// TIA Portal V18 export
FUNCTION "Function Selection HMI _Site_PB" : Void   // FC30, LAD
{ S7_Optimized_Access := 'TRUE' }
VERSION : 0.1
// stored: AutoNumber true, IsIECCheckEnabled false, SetENOAutomatically false, UDAEnableTagReadback false
   VAR_TEMP
      temp_unitsel : Int;
   END_VAR
   VAR_TEMP   // added for the SCL form of the ladder/FBD networks
      _w1 : Bool;
      _w2 : Bool;
   END_VAR
BEGIN

REGION Network 1: No functions selected
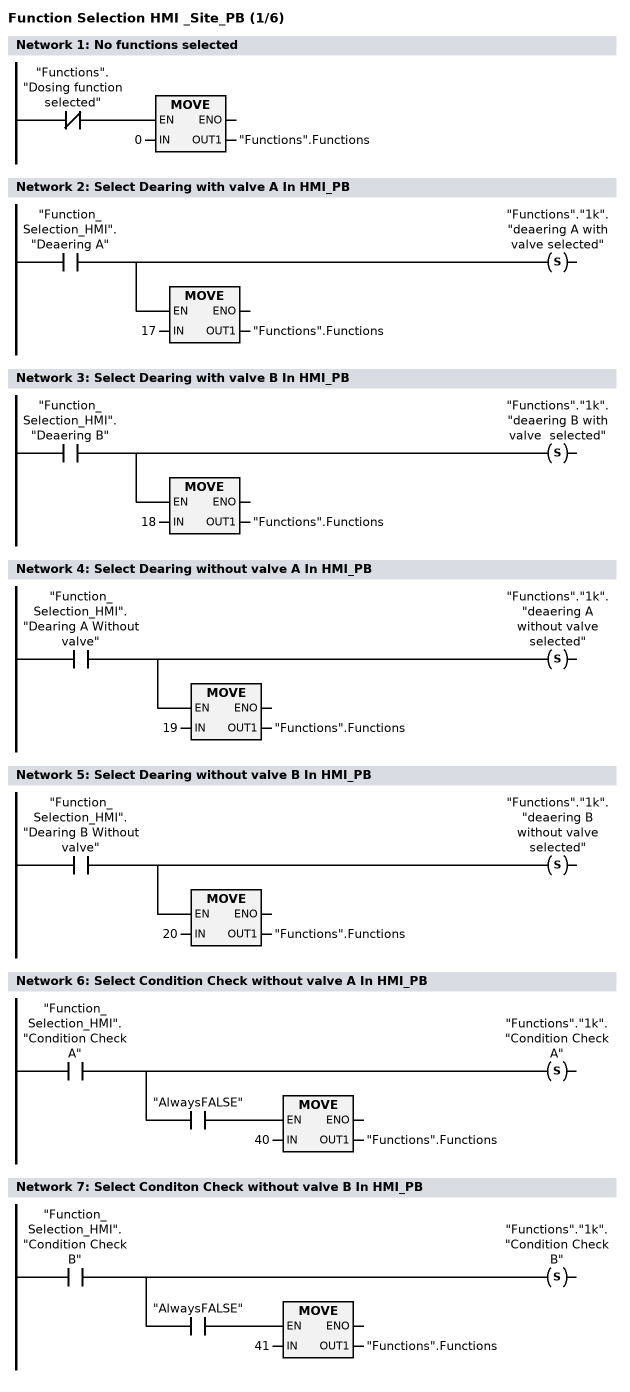
   RUNG wire#powerrail
      I_Contact( "Functions"."Dosing function selected" )
      Move(in := 0, out1 => "Functions".Functions)
   END_RUNG
   // the same network as SCL:
   IF NOT "Functions"."Dosing function selected" THEN "Functions".Functions := 0; END_IF;
END_REGION

REGION Network 2: Select Dearing with valve A In HMI_PB
   RUNG wire#powerrail
      Contact( "Function_Selection_HMI"."Deaering A" )
      wire#w1
      S_Coil( "Functions"."1k"."deaering A with valve selected" )
   END_RUNG
   RUNG wire#w1
      Move(in := 17, out1 => "Functions".Functions)
   END_RUNG
   // the same network as SCL:
   IF "Function_Selection_HMI"."Deaering A" THEN
       "Functions"."1k"."deaering A with valve selected" := TRUE;
       "Functions".Functions := 17;
   END_IF;
END_REGION

REGION Network 3: Select Dearing with valve B In HMI_PB
   RUNG wire#powerrail
      Contact( "Function_Selection_HMI"."Deaering B" )
      wire#w1
      S_Coil( "Functions"."1k"."deaering B with valve  selected" )
   END_RUNG
   RUNG wire#w1
      Move(in := 18, out1 => "Functions".Functions)
   END_RUNG
   // the same network as SCL:
   IF "Function_Selection_HMI"."Deaering B" THEN
       "Functions"."1k"."deaering B with valve  selected" := TRUE;
       "Functions".Functions := 18;
   END_IF;
END_REGION

REGION Network 4: Select Dearing without valve A In HMI_PB
   RUNG wire#powerrail
      Contact( "Function_Selection_HMI"."Dearing A Without valve" )
      wire#w1
      S_Coil( "Functions"."1k"."deaering A without valve selected" )
   END_RUNG
   RUNG wire#w1
      Move(in := 19, out1 => "Functions".Functions)
   END_RUNG
   // the same network as SCL:
   IF "Function_Selection_HMI"."Dearing A Without valve" THEN
       "Functions"."1k"."deaering A without valve selected" := TRUE;
       "Functions".Functions := 19;
   END_IF;
END_REGION

REGION Network 5: Select Dearing without valve B In HMI_PB
   RUNG wire#powerrail
      Contact( "Function_Selection_HMI"."Dearing B Without valve" )
      wire#w1
      S_Coil( "Functions"."1k"."deaering B without valve  selected" )
   END_RUNG
   RUNG wire#w1
      Move(in := 20, out1 => "Functions".Functions)
   END_RUNG
   // the same network as SCL:
   IF "Function_Selection_HMI"."Dearing B Without valve" THEN
       "Functions"."1k"."deaering B without valve  selected" := TRUE;
       "Functions".Functions := 20;
   END_IF;
END_REGION

REGION Network 6: Select Condition Check without valve A In HMI_PB
   RUNG wire#powerrail
      Contact( "Function_Selection_HMI"."Condition Check A" )
      wire#w1
      S_Coil( "Functions"."1k"."Condition Check A" )
   END_RUNG
   RUNG wire#w1
      Contact( "AlwaysFALSE" )
      Move(in := 40, out1 => "Functions".Functions)
   END_RUNG
   // the same network as SCL:
   IF "Function_Selection_HMI"."Condition Check A" THEN "Functions"."1k"."Condition Check A" := TRUE; END_IF;
   IF "Function_Selection_HMI"."Condition Check A" AND "AlwaysFALSE" THEN
       "Functions".Functions := 40;
   END_IF;
END_REGION

REGION Network 7: Select Conditon Check without valve B In HMI_PB
   RUNG wire#powerrail
      Contact( "Function_Selection_HMI"."Condition Check B" )
      wire#w1
      S_Coil( "Functions"."1k"."Condition Check B" )
   END_RUNG
   RUNG wire#w1
      Contact( "AlwaysFALSE" )
      Move(in := 41, out1 => "Functions".Functions)
   END_RUNG
   // the same network as SCL:
   IF "Function_Selection_HMI"."Condition Check B" THEN "Functions"."1k"."Condition Check B" := TRUE; END_IF;
   IF "Function_Selection_HMI"."Condition Check B" AND "AlwaysFALSE" THEN
       "Functions".Functions := 41;
   END_IF;
END_REGION

REGION Network 8: Select Recirculation A
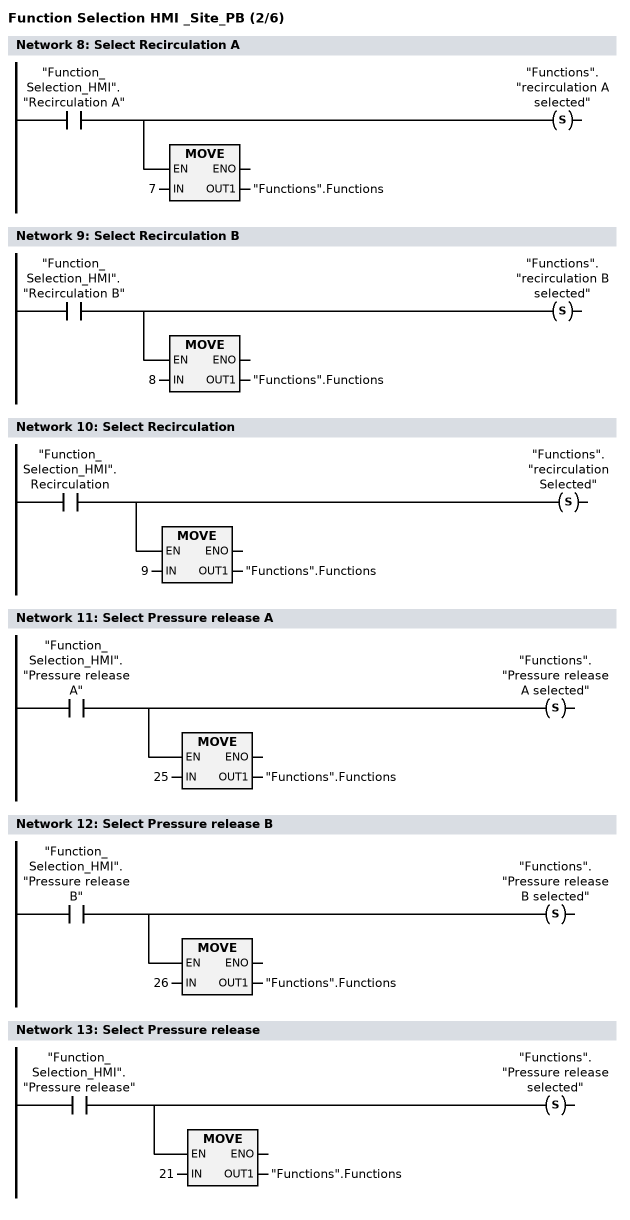
   RUNG wire#powerrail
      Contact( "Function_Selection_HMI"."Recirculation A" )
      wire#w1
      S_Coil( "Functions"."recirculation A selected" )
   END_RUNG
   RUNG wire#w1
      Move(in := 7, out1 => "Functions".Functions)
   END_RUNG
   // the same network as SCL:
   IF "Function_Selection_HMI"."Recirculation A" THEN
       "Functions"."recirculation A selected" := TRUE;
       "Functions".Functions := 7;
   END_IF;
END_REGION

REGION Network 9: Select Recirculation B
   RUNG wire#powerrail
      Contact( "Function_Selection_HMI"."Recirculation B" )
      wire#w1
      S_Coil( "Functions"."recirculation B selected" )
   END_RUNG
   RUNG wire#w1
      Move(in := 8, out1 => "Functions".Functions)
   END_RUNG
   // the same network as SCL:
   IF "Function_Selection_HMI"."Recirculation B" THEN
       "Functions"."recirculation B selected" := TRUE;
       "Functions".Functions := 8;
   END_IF;
END_REGION

REGION Network 10: Select Recirculation
   RUNG wire#powerrail
      Contact( "Function_Selection_HMI".Recirculation )
      wire#w1
      S_Coil( "Functions"."recirculation Selected" )
   END_RUNG
   RUNG wire#w1
      Move(in := 9, out1 => "Functions".Functions)
   END_RUNG
   // the same network as SCL:
   IF "Function_Selection_HMI".Recirculation THEN
       "Functions"."recirculation Selected" := TRUE;
       "Functions".Functions := 9;
   END_IF;
END_REGION

REGION Network 11: Select Pressure release A
   RUNG wire#powerrail
      Contact( "Function_Selection_HMI"."Pressure release A" )
      wire#w1
      S_Coil( "Functions"."Pressure release A selected" )
   END_RUNG
   RUNG wire#w1
      Move(in := 25, out1 => "Functions".Functions)
   END_RUNG
   // the same network as SCL:
   IF "Function_Selection_HMI"."Pressure release A" THEN
       "Functions"."Pressure release A selected" := TRUE;
       "Functions".Functions := 25;
   END_IF;
END_REGION

REGION Network 12: Select Pressure release B
   RUNG wire#powerrail
      Contact( "Function_Selection_HMI"."Pressure release B" )
      wire#w1
      S_Coil( "Functions"."Pressure release B selected" )
   END_RUNG
   RUNG wire#w1
      Move(in := 26, out1 => "Functions".Functions)
   END_RUNG
   // the same network as SCL:
   IF "Function_Selection_HMI"."Pressure release B" THEN
       "Functions"."Pressure release B selected" := TRUE;
       "Functions".Functions := 26;
   END_IF;
END_REGION

REGION Network 13: Select Pressure release
   RUNG wire#powerrail
      Contact( "Function_Selection_HMI"."Pressure release" )
      wire#w1
      S_Coil( "Functions"."Pressure release selected" )
   END_RUNG
   RUNG wire#w1
      Move(in := 21, out1 => "Functions".Functions)
   END_RUNG
   // the same network as SCL:
   IF "Function_Selection_HMI"."Pressure release" THEN
       "Functions"."Pressure release selected" := TRUE;
       "Functions".Functions := 21;
   END_IF;
END_REGION

REGION Network 14: Select shot metering
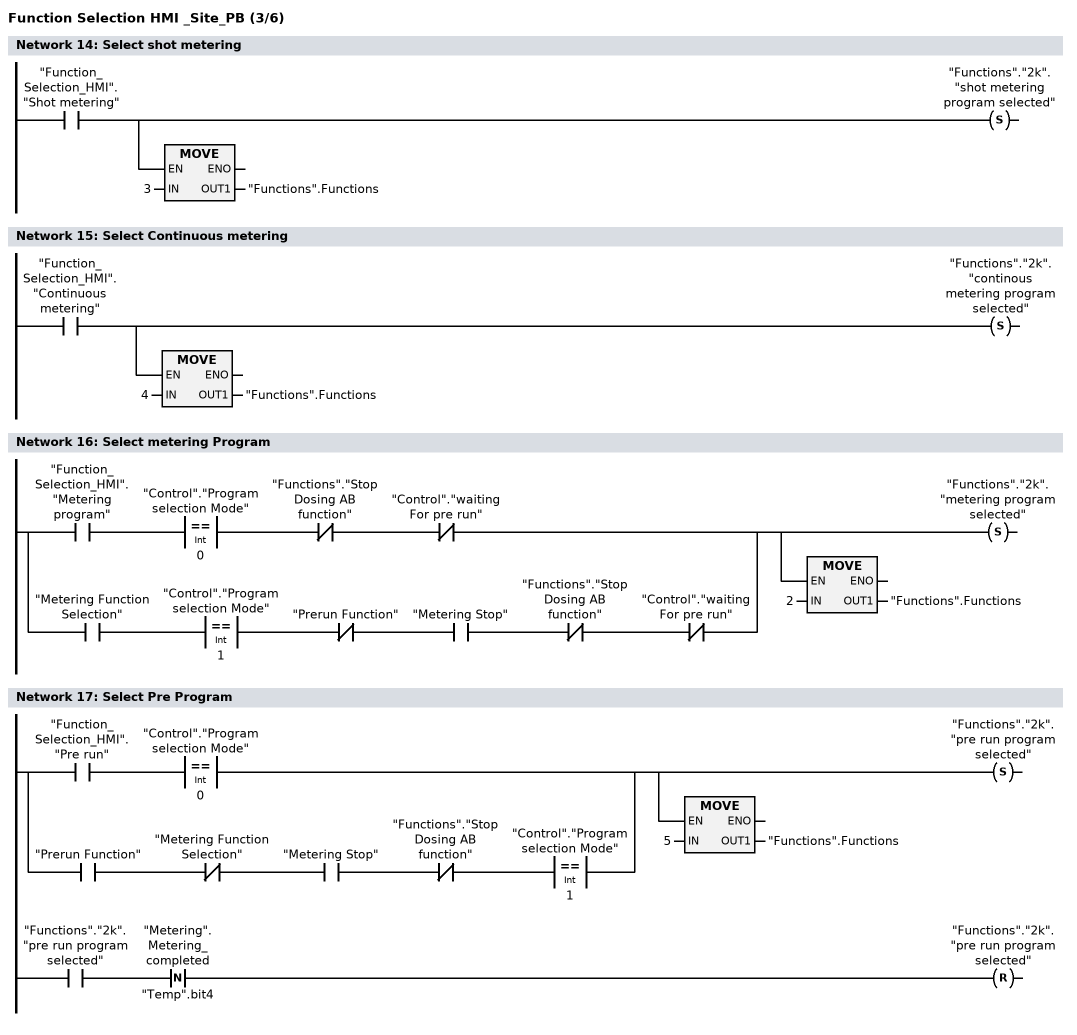
   RUNG wire#powerrail
      Contact( "Function_Selection_HMI"."Shot metering" )
      wire#w1
      S_Coil( "Functions"."2k"."shot metering program selected" )
   END_RUNG
   RUNG wire#w1
      Move(in := 3, out1 => "Functions".Functions)
   END_RUNG
   // the same network as SCL:
   IF "Function_Selection_HMI"."Shot metering" THEN
       "Functions"."2k"."shot metering program selected" := TRUE;
       "Functions".Functions := 3;
   END_IF;
END_REGION

REGION Network 15: Select Continuous metering
   RUNG wire#powerrail
      Contact( "Function_Selection_HMI"."Continuous metering" )
      wire#w1
      S_Coil( "Functions"."2k"."continous metering program selected" )
   END_RUNG
   RUNG wire#w1
      Move(in := 4, out1 => "Functions".Functions)
   END_RUNG
   // the same network as SCL:
   IF "Function_Selection_HMI"."Continuous metering" THEN
       "Functions"."2k"."continous metering program selected" := TRUE;
       "Functions".Functions := 4;
   END_IF;
END_REGION

REGION Network 16: Select metering Program
   RUNG wire#powerrail
      Contact( "Function_Selection_HMI"."Metering program" )
      { S7_Templates := "SrcType := Int" } EQ_Contact(in1 := "Control"."Program selection Mode", in2 := 0)
      I_Contact( "Functions"."Stop Dosing AB function" )
      I_Contact( "Control"."waiting For pre run" )
      wire#w1
      S_Coil( "Functions"."2k"."metering program selected" )
   END_RUNG
   RUNG wire#powerrail
      Contact( "Metering Function Selection" )
      { S7_Templates := "SrcType := Int" } EQ_Contact(in1 := "Control"."Program selection Mode", in2 := 1)
      I_Contact( "Prerun Function" )
      Contact( "Metering Stop" )
      I_Contact( "Functions"."Stop Dosing AB function" )
      I_Contact( "Control"."waiting For pre run" )
   END_RUNG wire#w1
   RUNG wire#w1
      Move(in := 2, out1 => "Functions".Functions)
   END_RUNG
   // the same network as SCL:
   IF ("Function_Selection_HMI"."Metering program" AND ("Control"."Program selection Mode" = 0) AND NOT "Functions"."Stop Dosing AB function" AND NOT "Control"."waiting For pre run") OR ("Metering Function Selection" AND ("Control"."Program selection Mode" = 1) AND NOT "Prerun Function" AND "Metering Stop" AND NOT "Functions"."Stop Dosing AB function" AND NOT "Control"."waiting For pre run") THEN
       "Functions"."2k"."metering program selected" := TRUE;
       "Functions".Functions := 2;
   END_IF;
END_REGION

REGION Network 17: Select Pre Program
   RUNG wire#powerrail
      Contact( "Function_Selection_HMI"."Pre run" )
      { S7_Templates := "SrcType := Int" } EQ_Contact(in1 := "Control"."Program selection Mode", in2 := 0)
      wire#w1
      S_Coil( "Functions"."2k"."pre run program selected" )
   END_RUNG
   RUNG wire#powerrail
      Contact( "Prerun Function" )
      I_Contact( "Metering Function Selection" )
      Contact( "Metering Stop" )
      I_Contact( "Functions"."Stop Dosing AB function" )
      { S7_Templates := "SrcType := Int" } EQ_Contact(in1 := "Control"."Program selection Mode", in2 := 1)
   END_RUNG wire#w1
   RUNG wire#w1
      Move(in := 5, out1 => "Functions".Functions)
   END_RUNG
   RUNG wire#powerrail
      Contact( "Functions"."2k"."pre run program selected" )
      N_Contact(operand := "Metering".Metering_completed, bit := "Temp".bit4)
      R_Coil( "Functions"."2k"."pre run program selected" )
   END_RUNG
   // the same network as SCL:
   IF ("Function_Selection_HMI"."Pre run" AND ("Control"."Program selection Mode" = 0)) OR ("Prerun Function" AND NOT "Metering Function Selection" AND "Metering Stop" AND NOT "Functions"."Stop Dosing AB function" AND ("Control"."Program selection Mode" = 1)) THEN
       "Functions"."2k"."pre run program selected" := TRUE;
       "Functions".Functions := 5;
   END_IF;
   #_w1 := "Functions"."2k"."pre run program selected" AND NOT "Metering".Metering_completed AND "Temp".bit4;   // falling edge of "Metering".Metering_completed
   "Temp".bit4 := "Metering".Metering_completed;
   IF #_w1 THEN "Functions"."2k"."pre run program selected" := FALSE; END_IF;
END_REGION

REGION Network 18: Select Ratio Program
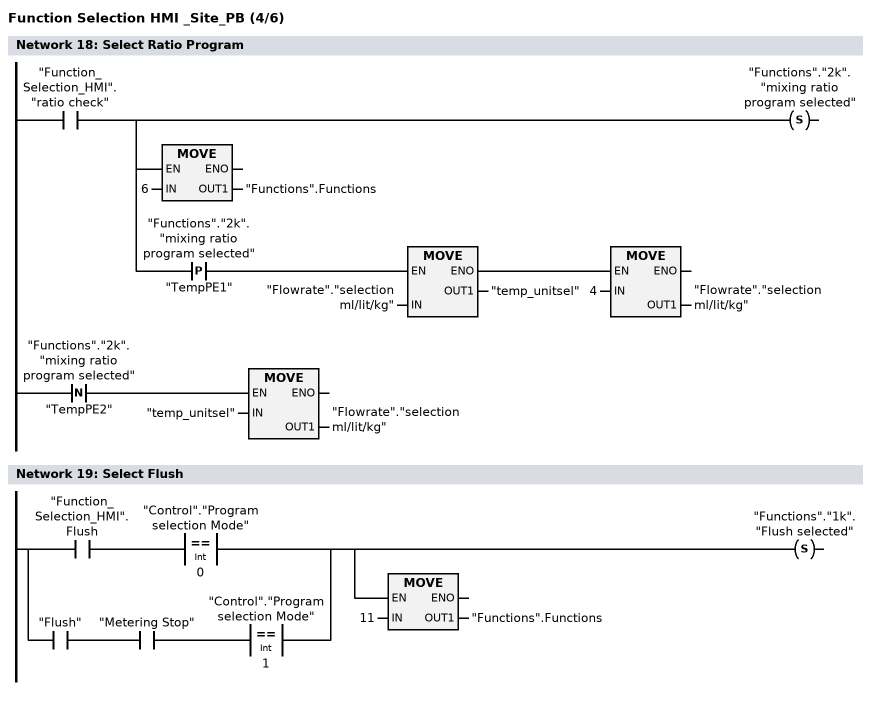
   RUNG wire#powerrail
      Contact( "Function_Selection_HMI"."ratio check" )
      wire#w1
      S_Coil( "Functions"."2k"."mixing ratio program selected" )
   END_RUNG
   RUNG wire#w1
      Move(in := 6, out1 => "Functions".Functions)
   END_RUNG
   RUNG wire#w1
      P_Contact(operand := "Functions"."2k"."mixing ratio program selected", bit := "TempPE1")
      Move(in := "Flowrate"."selection ml/lit/kg", out1 => "temp_unitsel")
      Move(in := 4, out1 => "Flowrate"."selection ml/lit/kg")
   END_RUNG
   RUNG wire#powerrail
      N_Contact(operand := "Functions"."2k"."mixing ratio program selected", bit := "TempPE2")
      Move(in := "temp_unitsel", out1 => "Flowrate"."selection ml/lit/kg")
   END_RUNG
   // the same network as SCL:
   IF "Function_Selection_HMI"."ratio check" THEN
       "Functions"."2k"."mixing ratio program selected" := TRUE;
       "Functions".Functions := 6;
   END_IF;
   #_w1 := "Function_Selection_HMI"."ratio check" AND "Functions"."2k"."mixing ratio program selected" AND NOT "TempPE1";   // rising edge of "Functions"."2k"."mixing ratio program selected"
   "TempPE1" := "Functions"."2k"."mixing ratio program selected";
   IF #_w1 THEN
       "temp_unitsel" := "Flowrate"."selection ml/lit/kg";
       "Flowrate"."selection ml/lit/kg" := 4;
   END_IF;
   #_w2 := NOT "Functions"."2k"."mixing ratio program selected" AND "TempPE2";   // falling edge of "Functions"."2k"."mixing ratio program selected"
   "TempPE2" := "Functions"."2k"."mixing ratio program selected";
   IF #_w2 THEN "Flowrate"."selection ml/lit/kg" := "temp_unitsel"; END_IF;
END_REGION

REGION Network 19: Select Flush
   RUNG wire#powerrail
      Contact( "Function_Selection_HMI".Flush )
      { S7_Templates := "SrcType := Int" } EQ_Contact(in1 := "Control"."Program selection Mode", in2 := 0)
      wire#w1
      S_Coil( "Functions"."1k"."Flush selected" )
   END_RUNG
   RUNG wire#powerrail
      Contact( "Flush" )
      Contact( "Metering Stop" )
      { S7_Templates := "SrcType := Int" } EQ_Contact(in1 := "Control"."Program selection Mode", in2 := 1)
   END_RUNG wire#w1
   RUNG wire#w1
      Move(in := 11, out1 => "Functions".Functions)
   END_RUNG
   // the same network as SCL:
   IF ("Function_Selection_HMI".Flush AND ("Control"."Program selection Mode" = 0)) OR ("Flush" AND "Metering Stop" AND ("Control"."Program selection Mode" = 1)) THEN
       "Functions"."1k"."Flush selected" := TRUE;
       "Functions".Functions := 11;
   END_IF;
END_REGION

REGION Network 20: Select Flush during potlife
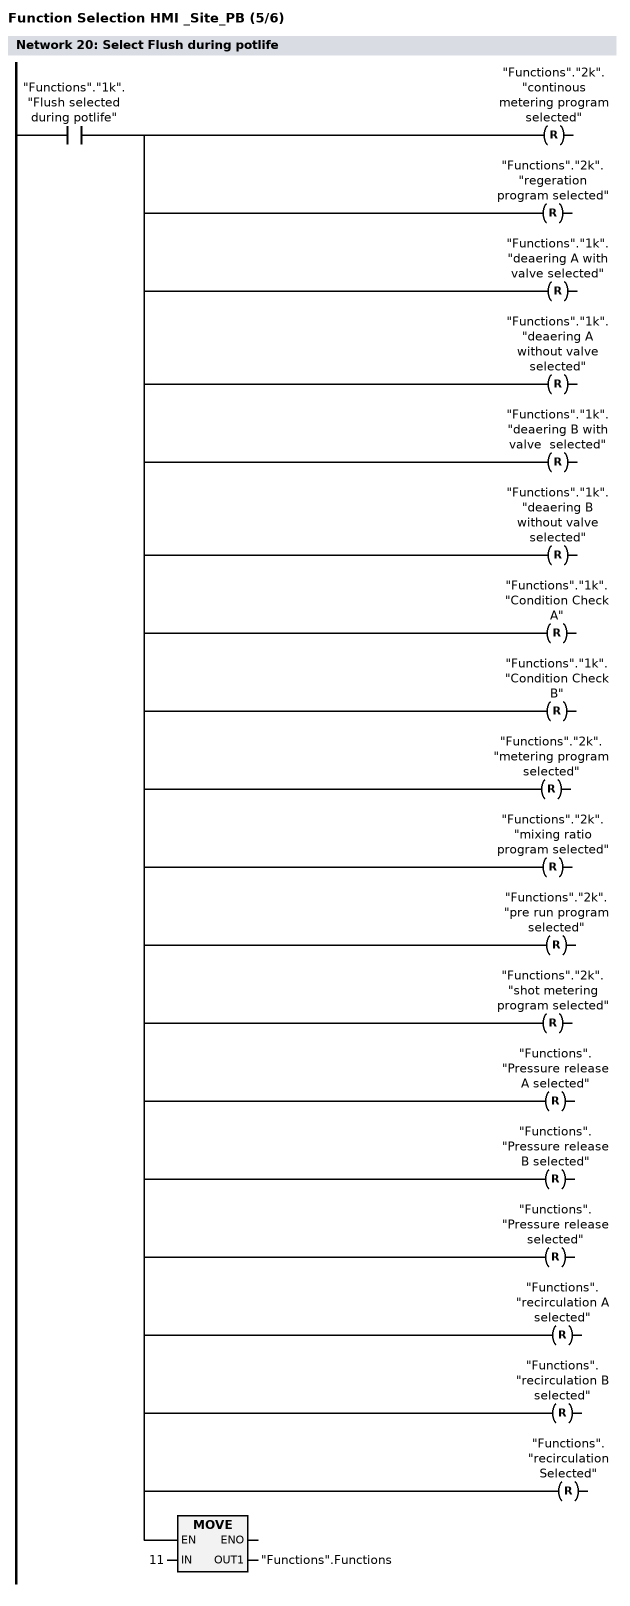
   RUNG wire#powerrail
      Contact( "Functions"."1k"."Flush selected during potlife" )
      wire#w1
      R_Coil( "Functions"."2k"."continous metering program selected" )
   END_RUNG
   RUNG wire#w1
      R_Coil( "Functions"."2k"."regeration program selected" )
   END_RUNG
   RUNG wire#w1
      R_Coil( "Functions"."1k"."deaering A with valve selected" )
   END_RUNG
   RUNG wire#w1
      R_Coil( "Functions"."1k"."deaering A without valve selected" )
   END_RUNG
   RUNG wire#w1
      R_Coil( "Functions"."1k"."deaering B with valve  selected" )
   END_RUNG
   RUNG wire#w1
      R_Coil( "Functions"."1k"."deaering B without valve  selected" )
   END_RUNG
   RUNG wire#w1
      R_Coil( "Functions"."1k"."Condition Check A" )
   END_RUNG
   RUNG wire#w1
      R_Coil( "Functions"."1k"."Condition Check B" )
   END_RUNG
   RUNG wire#w1
      R_Coil( "Functions"."2k"."metering program selected" )
   END_RUNG
   RUNG wire#w1
      R_Coil( "Functions"."2k"."mixing ratio program selected" )
   END_RUNG
   RUNG wire#w1
      R_Coil( "Functions"."2k"."pre run program selected" )
   END_RUNG
   RUNG wire#w1
      R_Coil( "Functions"."2k"."shot metering program selected" )
   END_RUNG
   RUNG wire#w1
      R_Coil( "Functions"."Pressure release A selected" )
   END_RUNG
   RUNG wire#w1
      R_Coil( "Functions"."Pressure release B selected" )
   END_RUNG
   RUNG wire#w1
      R_Coil( "Functions"."Pressure release selected" )
   END_RUNG
   RUNG wire#w1
      R_Coil( "Functions"."recirculation A selected" )
   END_RUNG
   RUNG wire#w1
      R_Coil( "Functions"."recirculation B selected" )
   END_RUNG
   RUNG wire#w1
      R_Coil( "Functions"."recirculation Selected" )
   END_RUNG
   RUNG wire#w1
      Move(in := 11, out1 => "Functions".Functions)
   END_RUNG
   // the same network as SCL:
   IF "Functions"."1k"."Flush selected during potlife" THEN
       "Functions"."2k"."continous metering program selected" := FALSE;
       "Functions"."2k"."regeration program selected" := FALSE;
       "Functions"."1k"."deaering A with valve selected" := FALSE;
       "Functions"."1k"."deaering A without valve selected" := FALSE;
       "Functions"."1k"."deaering B with valve  selected" := FALSE;
       "Functions"."1k"."deaering B without valve  selected" := FALSE;
       "Functions"."1k"."Condition Check A" := FALSE;
       "Functions"."1k"."Condition Check B" := FALSE;
       "Functions"."2k"."metering program selected" := FALSE;
       "Functions"."2k"."mixing ratio program selected" := FALSE;
       "Functions"."2k"."pre run program selected" := FALSE;
       "Functions"."2k"."shot metering program selected" := FALSE;
       "Functions"."Pressure release A selected" := FALSE;
       "Functions"."Pressure release B selected" := FALSE;
       "Functions"."Pressure release selected" := FALSE;
       "Functions"."recirculation A selected" := FALSE;
       "Functions"."recirculation B selected" := FALSE;
       "Functions"."recirculation Selected" := FALSE;
       "Functions".Functions := 11;
   END_IF;
END_REGION

REGION Network 21: regeneration selected
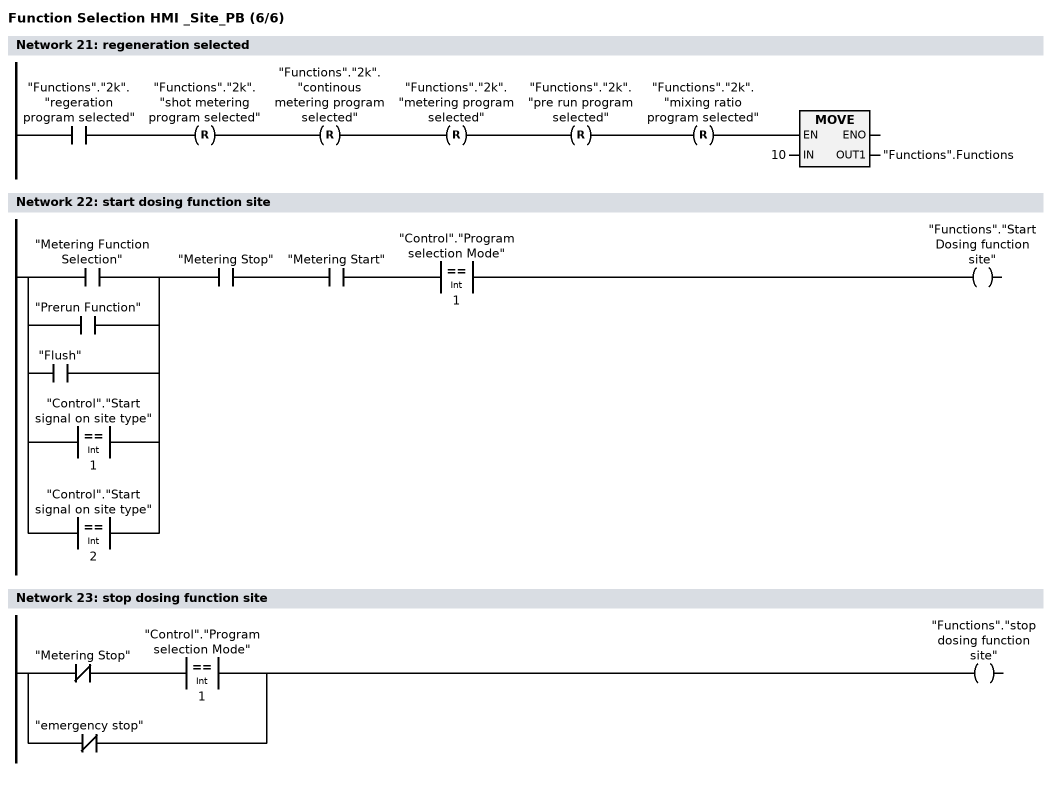
   RUNG wire#powerrail
      Contact( "Functions"."2k"."regeration program selected" )
      R_Coil( "Functions"."2k"."shot metering program selected" )
      R_Coil( "Functions"."2k"."continous metering program selected" )
      R_Coil( "Functions"."2k"."metering program selected" )
      R_Coil( "Functions"."2k"."pre run program selected" )
      R_Coil( "Functions"."2k"."mixing ratio program selected" )
      Move(in := 10, out1 => "Functions".Functions)
   END_RUNG
   // the same network as SCL:
   IF "Functions"."2k"."regeration program selected" THEN
       "Functions"."2k"."shot metering program selected" := FALSE;
       "Functions"."2k"."continous metering program selected" := FALSE;
       "Functions"."2k"."metering program selected" := FALSE;
       "Functions"."2k"."pre run program selected" := FALSE;
       "Functions"."2k"."mixing ratio program selected" := FALSE;
       "Functions".Functions := 10;
   END_IF;
END_REGION

REGION Network 22: start dosing function site
   RUNG wire#powerrail
      Contact( "Metering Function Selection" )
      wire#w1
      Contact( "Metering Stop" )
      Contact( "Metering Start" )
      { S7_Templates := "SrcType := Int" } EQ_Contact(in1 := "Control"."Program selection Mode", in2 := 1)
      Coil( "Functions"."Start Dosing function site" )
   END_RUNG
   RUNG wire#powerrail
      Contact( "Prerun Function" )
   END_RUNG wire#w1
   RUNG wire#powerrail
      Contact( "Flush" )
   END_RUNG wire#w1
   RUNG wire#powerrail
      { S7_Templates := "SrcType := Int" } EQ_Contact(in1 := "Control"."Start signal on site type", in2 := 1)
   END_RUNG wire#w1
   RUNG wire#powerrail
      { S7_Templates := "SrcType := Int" } EQ_Contact(in1 := "Control"."Start signal on site type", in2 := 2)
   END_RUNG wire#w1
   // the same network as SCL:
   "Functions"."Start Dosing function site" := ("Metering Function Selection" OR "Prerun Function" OR "Flush" OR ("Control"."Start signal on site type" = 1) OR ("Control"."Start signal on site type" = 2)) AND "Metering Stop" AND "Metering Start" AND ("Control"."Program selection Mode" = 1);
END_REGION

REGION Network 23: stop dosing function site
   RUNG wire#powerrail
      I_Contact( "Metering Stop" )
      { S7_Templates := "SrcType := Int" } EQ_Contact(in1 := "Control"."Program selection Mode", in2 := 1)
      wire#w1
      Coil( "Functions"."stop dosing function site" )
   END_RUNG
   RUNG wire#powerrail
      I_Contact( "emergency stop" )
   END_RUNG wire#w1
   // the same network as SCL:
   "Functions"."stop dosing function site" := (NOT "Metering Stop" AND ("Control"."Program selection Mode" = 1)) OR NOT "emergency stop";
END_REGION
END_FUNCTION
